TYPE ST_Thickness :
STRUCT
T_start :BOOL;
T_finish :BOOL;
T_OK     :BOOL;	
T_NG     :BOOL;
END_STRUCT
END_TYPE

(* stored: Version 1.1.0.1, ProductVersion 3.1.4024.9
   DUT ST_Thickness: Id {ed9fc533-0490-4f0d-be29-8641004d6050} *)
